(* CODESYS project Siri 18-4-2020.project
   Title: Prova ModbusTCP esclavo
   Version: 0.0.0.0
   Author: francisco.florensa

Project tree, tasks and I/O mapping:
  MyController : TM241CEC24R, Schneider Electric, order no. TM241CEC24R, version 4.0.6.18
    application Application
      task MAST (cyclic, interval 20 ms, priority 15, watchdog 100 ms x 1) calls POU
      task VISU_TASK (cyclic, interval 100 ms, priority 30) calls VisuElems.Visu_Prg
      global variables GVL
      program POU [LD]
      visualisation Caves_tancs_tiratge
      image pool ImagePool
      Symbols
    DI : Digital Inputs, Schneider Electric, version 4.0.6.18
        input  iwDI_IW0 : WORD  // IW0
        input  ibDI_IB1 : BYTE  // IB1
    DQ : Digital Outputs, Schneider Electric, version 4.0.6.18
        output xq_salida0 : BOOL  // QW0.Q0
        output xq_salida1 : BOOL  // QW0.Q1
        output xq_salida2 : BOOL  // QW0.Q2
        output xq_salida_rele3 : BOOL  // QW0.Q3
        output xq_salida_rele4 : BOOL  // QW0.Q4
        output qbDQ_QB1 : BYTE  // QB1
        unmapped channels: QW0
    Counters : Counters, Schneider Electric, version 4.0.6.18
    Pulse_Generators : Pulse Generators, Schneider Electric, version 4.0.6.18
    Cartridge_1 : Cartridge, Schneider Electric, version 4.0.6.18
    IO_Bus : IO bus - TM3, Schneider Electric, version 4.0.6.18
    COM_Bus : COM bus, Schneider Electric, version 4.0.6.18
    Ethernet_1 : Ethernet Network, Schneider Electric, version 4.0.6.18
        settings: IPAddress = [192, 168, 1, 58]; SubnetMask = [255, 255, 255, 0]; GatewayAddress = [192, 168, 1, 1]; WebServer = TRUE; FTP Server = TRUE; SoMachine Protocol = TRUE; Modbus Server = TRUE; NetManage Protocol = TRUE; SNMP protocol = TRUE; Enable Routing = FALSE; WebVisu protocol = TRUE; DHCP Server Active = FALSE
    Serial_Line_1 : Serial line, Schneider Electric, version 4.0.6.18
      SoMachine_Network_Manager : SoMachine-Network Manager, Schneider Electric, version 4.0.0.2
    Serial_Line_2 : Serial line, Schneider Electric, version 4.0.6.18
      Modbus_Manager : Modbus Manager, Schneider Electric, version 4.0.0.2
    CAN_1 : CANopen bus, Schneider Electric, version 4.0.6.18
  HMISCUxA5 : HMISCUxA5, Schneider Electric, order no. HMISCUxA5, version 3.5.3.59
    application Application
      task MAST (cyclic, interval 20 ms, priority 15, watchdog 100 ms x 1) calls nothing
      global variables GVL
    HMI Application
    Ethernet
      SoMachine_Network_Manager2 : SoMachine-Network Manager, Schneider Electric, version 4.0.0.2
    CAN
    Funciones incorporadas
      ES : ES, Schneider Electric, order no. IO, version 3.5.3.59
          input  iwES_Entrada : WORD  // In
          output qwES_Salida : WORD  // Out
      PTO_PWM : PTO_PWM, Schneider Electric, order no. PTO_PWM, version 3.5.3.59
      HSC : HSC, Schneider Electric, order no. HSC, version 3.5.3.59
    COM1
      SoMachine_Network_Manager1 : SoMachine-Network Manager, Schneider Electric, version 4.0.0.2
    USB
      SoMachine_Network_Manager3 : SoMachine-Network Manager, Schneider Electric, version 4.0.0.2
  text list GlobalTextList
  5ce3da45-db07-42e7-a21c-a00fff4ed8f6|C:\Users\francisco.florensa\Documents\Marketing\Punts de venda\Vilanova\Caves Castelo de Pedregosa\caves.png
  Vijeo Designer Project Container Data
  Vijeo Designer Project Container
*)

// MyController/Application/GVL
VAR_GLOBAL
	var0 AT %MW0: INT;
	var1 AT %MW1: INT;
	var2 AT %MW2: INT;
	var3 AT %MW3: INT;
	var4 AT %MW4: INT;
	var5 AT %MW5: INT;
	var6 AT %MW6: INT;
	var7 AT %MW7: INT;
	var8 AT %MW8: INT;
	var9 AT %MW9: INT;
	BYTE_AS_BIT_0: BYTE_AS_BIT;
	WORD_AS_BIT_0: WORD_AS_BIT;
END_VAR

// HMISCUxA5/Application/GVL
VAR_GLOBAL
END_VAR

// MyController/Application/POU
PROGRAM POU
VAR
	i_sinusoidal: INT;
	
	i_peso AT %MW0: INT;
	GEN0: GEN;
	i_peso1 AT %QW2: INT;
	i_peso2 AT %QW3: INT;
	
END_VAR

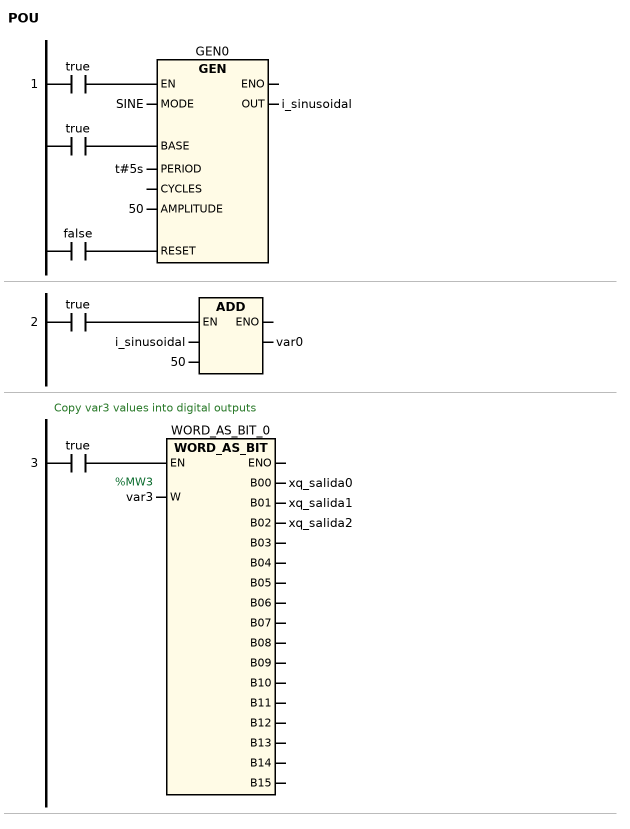
// NETWORK 1
IF true THEN
    GEN0(MODE := SINE, BASE := true, PERIOD := t#5s, AMPLITUDE := 50, RESET := false, OUT => i_sinusoidal); // GEN
END_IF

// NETWORK 2
//   var0: AT %MW0
IF true THEN var0 := i_sinusoidal + 50; END_IF

// NETWORK 3
// Copy var3 values into digital outputs
//   var3: AT %MW3
//   xq_salida0: DQ : Salida rápida, contrafase | AT %QX0.0
//   xq_salida1: DQ : Salida rápida, contrafase | AT %QX0.1
//   xq_salida2: DQ : Salida rápida, contrafase | AT %QX0.2
IF true THEN
    WORD_AS_BIT_0(W := var3, B00 => xq_salida0, B01 => xq_salida1, B02 => xq_salida2); // WORD_AS_BIT
END_IF

END_PROGRAM

// MyController/Application/Caves_tancs_tiratge
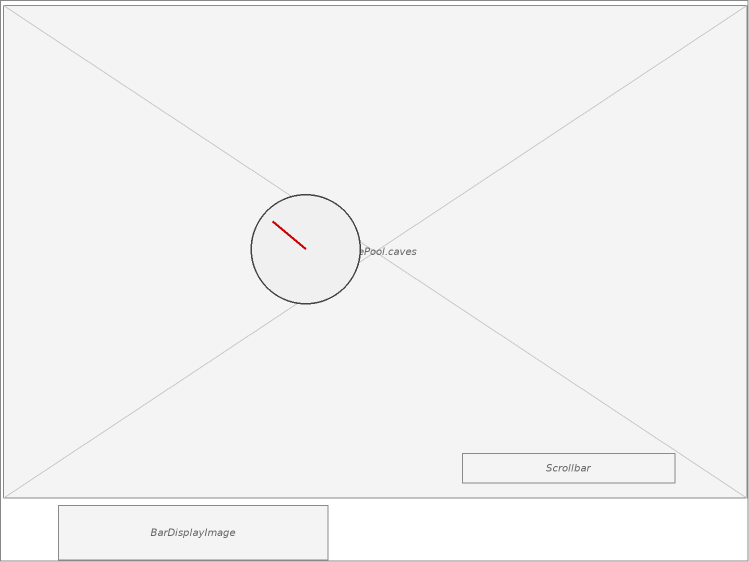
VISUALIZATION Caves_tancs_tiratge  // 749x562
    BarDisplayImage (58,505 270x55), value: var0, style: BarDisplayImage-Gray, scale format: %.1f, scale 0..100
    Image (3,5 744x493), image: ImagePool.caves
    Meter360 (247,194 117x110), value: var3, style: Meter-Meter360-Gray, scale format: %.1f, scale 0..100
    Scrollbar (462,453 213x30)
        p1057716461: var3
END_VISUALIZATION
